FUNCTION_BLOCK FB_ManualImplementation IMPLEMENTS  I_ManualImplementation
VAR_INPUT
		i_ManualControl : ARRAY[0..12,0..12] OF I_ManualControl;
END_VAR
VAR_OUTPUT
END_VAR
VAR
	i: INT;
	j: INT;
	k: INT;
	k_1: INT;
	bDosingPumpEnableVessels: BOOL;
	bDosingPumpEnableReactors: BOOL;

END_VAR

//=========================================================
// Instantiation Logic


	FOR k:=0 TO 10 DO
		FOR k_1 := 0 TO 10 DO
			IF i_ManualControl[k, k_1] <> 0 THEN
			THIS^.i_ManualControl[k, k_1] := i_ManualControl[k, k_1];
		END_IF	
		END_FOR
		
	END_FOR


//=========================================================
// Count Declaration Logic

	

//=========================================================
// Manual Logic
	
	//Manual Logic for Vessels.Valves
	
	FOR i:=0 TO 8 DO
		FOR j :=0 TO 7 DO
			IO.Vessels[i].Valves[j].Output :=i_ManualControl[i, j].
				M_RunValve(IO.Vessels[i].Valves[j].bStart);
		END_FOR
	END_FOR
	
	//Manual Logic for Vessels.Pumps
	
	FOR i:=0 TO 8 DO
		FOR j :=0 TO 1 DO
			//IO.Vessels[i].Pumps[j].nPulse := 6;
			IO.Vessels[i].Pumps[j].Output :=i_ManualControl[i,j].
				M_RunPump(IO.Vessels[i].Pumps[j].bStart,IO.Vessels[i].Pumps[j].nPulse);
			IF IO.Vessels[i].Pumps[j].bStart THEN
				bDosingPumpEnableVessels := TRUE;
			ELSE
				bDosingPumpEnableVessels := FALSE;
			END_IF
		END_FOR
	END_FOR
	
	//Manual Logic for Reactors.Valves
	
	FOR i:=0 TO 1 DO
		FOR j :=0 TO 7 DO
			IO.Reactors[i].Valves[j].Output :=i_ManualControl[9+i,j].
				M_RunValve(IO.Reactors[i].Valves[j].bStart);
		END_FOR
	END_FOR
	
	//Manual Logic for Reactors.Pumps
	
	FOR i:=0 TO 1 DO
		FOR j :=0 TO 1 DO
			IO.Reactors[i].Pumps[j].nPulse := 4;
			IO.Reactors[i].Pumps[j].Output :=i_ManualControl[9+i,j+1].
				M_RunPump(IO.Reactors[i].Pumps[j].bStart,IO.Reactors[i].Pumps[j].nPulse);
			IF IO.Reactors[i].Pumps[j].bStart THEN
				bDosingPumpEnableReactors := TRUE;
			ELSE
				bDosingPumpEnableReactors := FALSE;
			END_IF
		END_FOR
	END_FOR
	

//=========================================================
// Dosing Pump Enable Logic

IF IO.Vessels[0].Pumps[0].bStart OR IO.Vessels[0].Pumps[1].bStart
	OR IO.Vessels[1].Pumps[0].bStart OR IO.Vessels[1].Pumps[1].bStart
	OR IO.Vessels[2].Pumps[0].bStart OR IO.Vessels[2].Pumps[1].bStart
	OR IO.Vessels[3].Pumps[0].bStart OR IO.Vessels[3].Pumps[1].bStart
	OR IO.Vessels[4].Pumps[0].bStart OR IO.Vessels[4].Pumps[1].bStart
	OR IO.Vessels[5].Pumps[0].bStart OR IO.Vessels[5].Pumps[1].bStart
	OR IO.Vessels[6].Pumps[0].bStart OR IO.Vessels[6].Pumps[1].bStart
	OR IO.Vessels[7].Pumps[0].bStart OR IO.Vessels[7].Pumps[1].bStart
	OR IO.Vessels[8].Pumps[0].bStart OR IO.Vessels[8].Pumps[1].bStart
	OR IO.Reactors[0].Pumps[0].bStart OR IO.Reactors[0].Pumps[1].bStart
	OR IO.Reactors[1].Pumps[0].bStart OR IO.Reactors[1].Pumps[1].bStart THEN
	IO.PhysicalIO.DosingPumpEnable := TRUE;
ELSE
	IO.PhysicalIO.DosingPumpEnable := FALSE;

END_IF

//IF bDosingPumpEnableVessels OR bDosingPumpEnableReactors THEN

//END_IF

PROPERTY ipManualControl : ARRAY [0..12,0..12] OF I_ManualControl
GET
ipManualControl	:= i_ManualControl;
END_GET
END_PROPERTY

END_FUNCTION_BLOCK

(* stored: Version 1.1.0.1, ProductVersion 3.1.4024.9
   POU FB_ManualImplementation: Id {d5d23203-6915-44ea-a76c-32f9df040844}, SpecialFunc None
   Property ipManualControl: Id {ffd2fd39-3738-4c96-ac62-74dbe24a672c}
   Get Get: Id {b44032a2-4dc6-40ca-95bb-f854afed289d} *)
